PROGRAM prgFilterTesting
VAR
	t:LREAL;
	squareSignal:LREAL;
	valueAdd:LREAL:=0.01;
END_VAR

t:= t+valueAdd;

squareSignal:= SIN(t) + SIN(3*t)/3+ SIN(5*t)/5 + SIN(7*t)/7 + SIN(9*t)/9;

END_PROGRAM

(* stored: Version 1.1.0.1, ProductVersion 3.1.4024.12
   POU prgFilterTesting: Id {5d27849a-8e5a-4570-8dfc-86c2ad1a825b}, SpecialFunc None *)
